(* Logix 5000 project; controller Ex_2_14 Emulate 5570 rev 33.11; software revision 33.00 *)
// Pump well with one pump and two float switches

TASK MainTask (continuous, watchdog 500 ms) : MainProgram

MODULES
   Local : Emulate 5570 (ICP 4, rev 33.11)
END_MODULES

VAR_GLOBAL   (* controller tags *)
   LS1 : BOOL;   // Flot Switch LS1 (Top)
   LS2 : BOOL;   // Float Switch LS2 (Bottom)
   M1 : BOOL;   // Pump M1
   ONS_1 : BOOL;
END_VAR

PROGRAM MainProgram   (* main routine MainRoutine *)

ROUTINE MainRoutine   (* ladder *)
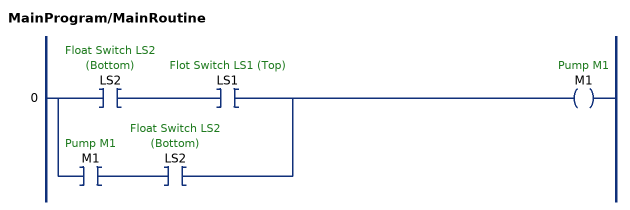
   0: [XIC(LS2) XIC(LS1) ,XIC(M1) XIC(LS2) ]OTE(M1);
END_ROUTINE
END_PROGRAM
